PROGRAM Door_Control
VAR
	State : INT :=0;
	Safety_Ok : BOOL;
END_VAR

CASE State OF
	0: 	//Idle state 
	Variables.Motor_Moving :=FALSE;
	//Wait for open button
	IF Variables.Button_Open THEN
		State :=10;
	END_IF
	
	10:	// Opening
	Safety_Ok := Safety(Variables.Safety_Sensor); // Check if it is safe
	IF Safety_OK = TRUE THEN
		Variables.Motor_Moving := TRUE; //Tell light task to turn on
		IF Variables.Sensor_Open THEN //Check if door reached the top
			State :=20;
		END_IF
	ELSE 
		State := 0; // Emergency stop
	END_IF
	
	20:	//Opened
	Variables.Motor_Moving :=FALSE;
	IF Variables.Button_Close THEN 	// Wait for close button
		State := 30;
	END_IF
	
	30: //Closing
	Safety_Ok := Safety(Variables.Safety_Sensor);
	IF Safety_Ok = TRUE THEN
		Variables.Motor_Moving := TRUE;
	
	IF Variables.Sensor_Close THEN //Check if door reached the bottom
		State :=0;
	END_IF
	ELSE
		State :=20; // If  there is an obstacle open
	END_IF
END_CASE

END_PROGRAM

(* stored: Version 1.1.0.1, ProductVersion 3.1.4024.15
   POU Door_Control: Id {f0de98ce-e84a-488c-b523-ef1d5b401766}, SpecialFunc None *)
